TYPE CNTOutputs :
STRUCT
	{attribute addProperty Name "Control"}
	Control AT %Q* : stCNTControl;
	{attribute addProperty Name "Set counter value"}
	SetCounterValue AT %Q* : UDINT;
END_STRUCT
END_TYPE

(* stored: Version 1.1.0.1, ProductVersion 3.1.4024.9
   DUT CNTOutputs: Id {e3214457-f9d5-0198-2f2a-92626eb3ed76} *)
